LIN {X 0,Y 62.579,Z 548.254,A -85,B 0,C 180,E1 -28523.551,E2 -28523.551} C_VEL
LIN {X 0,Y 62.497,Z 549.862,A -85,B 0,C 180,E1 -28529.999,E2 -28529.999} C_VEL
LIN {X 0,Y 63.288,Z 551.85,A -85,B 0,C 180,E1 -28542.831,E2 -28542.831} C_VEL
LIN {X 0,Y 66.65,Z 552.168,A -85,B 0,C 180,E1 -28554.947,E2 -28554.947} C_VEL
LIN {X 0,Y 69.259,Z 551.826,A -85,B 0,C 180,E1 -28560.488,E2 -28560.488} C_VEL
LIN {X 0,Y 76.403,Z 549.954,A -85,B 0,C 180,E1 -28570.083,E2 -28570.083} C_VEL
LIN {X 0,Y 85.273,Z 546.396,A -85,B 0,C 180,E1 -28577.881,E2 -28577.881} C_VEL
LIN {X 0,Y 92.403,Z 542.869,A -85,B 0,C 180,E1 -28582.523,E2 -28582.523} C_VEL
LIN {X 0,Y 100.815,Z 537.874,A -85,B 0,C 180,E1 -28586.776,E2 -28586.776} C_VEL
LIN {X 0,Y 107.932,Z 532.997,A -85,B 0,C 180,E1 -28589.629,E2 -28589.629} C_VEL
LIN {X 0,Y 116.859,Z 525.752,A -85,B 0,C 180,E1 -28592.508,E2 -28592.508} C_VEL
LIN {X 0,Y 124.397,Z 518.518,A -85,B 0,C 180,E1 -28594.681,E2 -28594.681} C_VEL
LIN {X 0,Y 132.226,Z 509.719,A -85,B 0,C 180,E1 -28596.471,E2 -28596.471} C_VEL
LIN {X 0,Y 138.528,Z 501.33,A -85,B 0,C 180,E1 -28597.802,E2 -28597.802} C_VEL
LIN {X 0,Y 144.119,Z 492.584,A -85,B 0,C 180,E1 -28598.849,E2 -28598.849} C_VEL
LIN {X 0,Y 148.94,Z 483.625,A -85,B 0,C 180,E1 -28599.691,E2 -28599.691} C_VEL
LIN {X 0,Y 153.773,Z 472.412,A -85,B 0,C 180,E1 -28600.425,E2 -28600.425} C_VEL
LIN {X 0,Y 157.625,Z 460.628,A -85,B 0,C 180,E1 -28600.964,E2 -28600.964} C_VEL
LIN {X 0,Y 159.421,Z 453.709,A -85,B 0,C 180,E1 -28601.223,E2 -28601.223} C_VEL
LIN {X 0,Y 158.999,Z 451.366,A -85,B 0,C 180,E1 -28604.293,E2 -28604.293} C_VEL
LIN {X 0,Y 158.718,Z 450.737,A -85,B 0,C 180,E1 -28607.21,E2 -28607.21} C_VEL
LIN {X 0,Y 158.819,Z 450.724,A -85,B 0,C 180,E1 -28610.207,E2 -28610.207} C_VEL
LIN {X 0,Y 159.185,Z 451.615,A -85,B 0,C 180,E1 -28613.027,E2 -28613.027} C_VEL
LIN {X 0,Y 159.452,Z 453.17,A -85,B 0,C 180,E1 -28614.943,E2 -28614.943} C_VEL
LIN {X 0,Y 156.119,Z 465.329,A -85,B 0,C 180,E1 -28615.461,E2 -28615.461} C_VEL
LIN {X 0,Y 155.317,Z 467.61,A -85,B 0,C 180,E1 -28615.586,E2 -28615.586} C_VEL
LIN {X 0,Y 153.244,Z 473.27,A -85,B 0,C 180,E1 -28615.697,E2 -28615.697} C_VEL
LIN {X 0,Y 149.004,Z 482.069,A -85,B 0,C 180,E1 -28615.23,E2 -28615.23} C_VEL
LIN {X 0,Y 144.136,Z 490.614,A -85,B 0,C 180,E1 -28614.827,E2 -28614.827} C_VEL
LIN {X 0,Y 140.951,Z 495.515,A -85,B 0,C 180,E1 -28615.081,E2 -28615.081} C_VEL
LIN {X 0,Y 133.801,Z 505.556,A -85,B 0,C 180,E1 -28616.364,E2 -28616.364} C_VEL
LIN {X 0,Y 126.592,Z 514.036,A -85,B 0,C 180,E1 -28617.856,E2 -28617.856} C_VEL
LIN {X 0,Y 119.48,Z 521.172,A -85,B 0,C 180,E1 -28619.505,E2 -28619.505} C_VEL
LIN {X 0,Y 110.749,Z 528.549,A -85,B 0,C 180,E1 -28621.864,E2 -28621.864} C_VEL
LIN {X 0,Y 104.495,Z 533.192,A -85,B 0,C 180,E1 -28623.857,E2 -28623.857} C_VEL
LIN {X 0,Y 95.637,Z 538.703,A -85,B 0,C 180,E1 -28627.224,E2 -28627.224} C_VEL
LIN {X 0,Y 86.174,Z 543.493,A -85,B 0,C 180,E1 -28631.857,E2 -28631.857} C_VEL
LIN {X 0,Y 80.245,Z 546.021,A -85,B 0,C 180,E1 -28635.55,E2 -28635.55} C_VEL
LIN {X 0,Y 71.071,Z 549.044,A -85,B 0,C 180,E1 -28643.302,E2 -28643.302} C_VEL
LIN {X 0,Y 65.17,Z 550.355,A -85,B 0,C 180,E1 -28650.377,E2 -28650.377} C_VEL
LIN {X 0,Y 61.39,Z 550.71,A -85,B 0,C 180,E1 -28656.74,E2 -28656.74} C_VEL
LIN {X 0,Y 56.246,Z 550.229,A -85,B 0,C 180,E1 -28671.336,E2 -28671.336} C_VEL
LIN {X 0,Y 54.695,Z 548.382,A -85,B 0,C 180,E1 -28684.091,E2 -28684.091} C_VEL
LIN {X 0,Y 55.311,Z 545.786,A -85,B 0,C 180,E1 -28695.279,E2 -28695.279} C_VEL
LIN {X 0,Y 57.758,Z 541.882,A -85,B 0,C 180,E1 -28706.513,E2 -28706.513} C_VEL
LIN {X 0,Y 61.564,Z 536.786,A -85,B 0,C 180,E1 -28716.556,E2 -28716.556} C_VEL
LIN {X 0,Y 65.869,Z 531.542,A -85,B 0,C 180,E1 -28723.891,E2 -28723.891} C_VEL
LIN {X 0,Y 71.007,Z 525.185,A -85,B 0,C 180,E1 -28730.269,E2 -28730.269} C_VEL
LIN {X 0,Y 76.87,Z 517.465,A -85,B 0,C 180,E1 -28735.74,E2 -28735.74} C_VEL
LIN {X 0,Y 82.172,Z 509.761,A -85,B 0,C 180,E1 -28739.735,E2 -28739.735} C_VEL
LIN {X 0,Y 88.054,Z 500.156,A -85,B 0,C 180,E1 -28743.28,E2 -28743.28} C_VEL
LIN {X 0,Y 93,Z 490.72,A -85,B 0,C 180,E1 -28745.851,E2 -28745.851} C_VEL
LIN {X 0,Y 97.459,Z 480.559,A -85,B 0,C 180,E1 -28747.91,E2 -28747.91} C_VEL
LIN {X 0,Y 101.142,Z 470.239,A -85,B 0,C 180,E1 -28749.46,E2 -28749.46} C_VEL
LIN {X 0,Y 104.051,Z 459.662,A -85,B 0,C 180,E1 -28750.645,E2 -28750.645} C_VEL
LIN {X 0,Y 106.272,Z 449.078,A -85,B 0,C 180,E1 -28751.401,E2 -28751.401} C_VEL
LIN {X 0,Y 108.672,Z 430.245,A -85,B 0,C 180,E1 -28752.234,E2 -28752.234} C_VEL
LIN {X 0,Y 109.348,Z 423.381,A -85,B 0,C 180,E1 -28752.568,E2 -28752.568} C_VEL
LIN {X 0,Y 105.848,Z 414.809,A -85,B 0,C 180,E1 -28756.918,E2 -28756.918} C_VEL
LIN {X 0,Y 103.278,Z 409.54,A -85,B 0,C 180,E1 -28760.478,E2 -28760.478} C_VEL
LIN {X 0,Y 100.68,Z 404.348,A -85,B 0,C 180,E1 -28764.837,E2 -28764.837} C_VEL
LIN {X 0,Y 98.374,Z 400.234,A -85,B 0,C 180,E1 -28769.578,E2 -28769.578} C_VEL
LIN {X 0,Y 96.622,Z 396.989,A -85,B 0,C 180,E1 -28774.494,E2 -28774.494} C_VEL
LIN {X 0,Y 94.923,Z 393.92,A -85,B 0,C 180,E1 -28782.772,E2 -28782.772} C_VEL
LIN {X 0,Y 94.765,Z 392.903,A -85,B 0,C 180,E1 -28786.033,E2 -28786.033} C_VEL
LIN {X 0,Y 95.042,Z 392.871,A -85,B 0,C 180,E1 -28792.896,E2 -28792.896} C_VEL
LIN {X 0,Y 95.334,Z 393.924,A -85,B 0,C 180,E1 -28795.422,E2 -28795.422} C_VEL
LIN {X 0,Y 97.049,Z 397.206,A -85,B 0,C 180,E1 -28802.516,E2 -28802.516} C_VEL
LIN {X 0,Y 99.172,Z 401.426,A -85,B 0,C 180,E1 -28807.955,E2 -28807.955} C_VEL
LIN {X 0,Y 101.485,Z 405.932,A -85,B 0,C 180,E1 -28812.443,E2 -28812.443} C_VEL
LIN {X 0,Y 104.35,Z 411.648,A -85,B 0,C 180,E1 -28816.885,E2 -28816.885} C_VEL
LIN {X 0,Y 107.69,Z 419.475,A -85,B 0,C 180,E1 -28821.321,E2 -28821.321} C_VEL
LIN {X 0,Y 109.234,Z 424.676,A -85,B 0,C 180,E1 -28823.327,E2 -28823.327} C_VEL
LIN {X 0,Y 106.575,Z 448.2,A -85,B 0,C 180,E1 -28824.439,E2 -28824.439} C_VEL
LIN {X 0,Y 104.902,Z 457.507,A -85,B 0,C 180,E1 -28825.063,E2 -28825.063} C_VEL
LIN {X 0,Y 102.29,Z 467.768,A -85,B 0,C 180,E1 -28825.997,E2 -28825.997} C_VEL
LIN {X 0,Y 98.791,Z 478.018,A -85,B 0,C 180,E1 -28827.22,E2 -28827.22} C_VEL
LIN {X 0,Y 94.568,Z 488.531,A -85,B 0,C 180,E1 -28829.163,E2 -28829.163} C_VEL
LIN {X 0,Y 90.311,Z 497.107,A -85,B 0,C 180,E1 -28831.126,E2 -28831.126} C_VEL
LIN {X 0,Y 84.902,Z 506.569,A -85,B 0,C 180,E1 -28834.128,E2 -28834.128} C_VEL
LIN {X 0,Y 79.778,Z 514.509,A -85,B 0,C 180,E1 -28837.546,E2 -28837.546} C_VEL
LIN {X 0,Y 73.749,Z 522.723,A -85,B 0,C 180,E1 -28842.392,E2 -28842.392} C_VEL
LIN {X 0,Y 68.428,Z 529.57,A -85,B 0,C 180,E1 -28848.117,E2 -28848.117} C_VEL
LIN {X 0,Y 64.698,Z 534.284,A -85,B 0,C 180,E1 -28853.311,E2 -28853.311} C_VEL
LIN {X 0,Y 60.049,Z 540.007,A -85,B 0,C 180,E1 -28862.085,E2 -28862.085} C_VEL
LIN {X 0,Y 57.018,Z 544.501,A -85,B 0,C 180,E1 -28872.052,E2 -28872.052} C_VEL
LIN {X 0,Y 55.536,Z 547.885,A -85,B 0,C 180,E1 -28882.729,E2 -28882.729} C_VEL
LIN {X 0,Y 55.399,Z 549.494,A -85,B 0,C 180,E1 -28889.999,E2 -28889.999} C_VEL
LIN {X 0,Y 56.369,Z 551.641,A -85,B 0,C 180,E1 -28904.439,E2 -28904.439} C_VEL
LIN {X 0,Y 60.26,Z 552.123,A -85,B 0,C 180,E1 -28917.807,E2 -28917.807} C_VEL
LIN {X 0,Y 66.907,Z 551.075,A -85,B 0,C 180,E1 -28929.067,E2 -28929.067} C_VEL
LIN {X 0,Y 71.12,Z 550.096,A -85,B 0,C 180,E1 -28933.767,E2 -28933.767} C_VEL
LIN {X 0,Y 80.688,Z 546.707,A -85,B 0,C 180,E1 -28941.619,E2 -28941.619} C_VEL
LIN {X 0,Y 87.713,Z 543.606,A -85,B 0,C 180,E1 -28945.885,E2 -28945.885} C_VEL
LIN {X 0,Y 97.13,Z 538.467,A -85,B 0,C 180,E1 -28950.258,E2 -28950.258} C_VEL
LIN {X 0,Y 106.057,Z 532.618,A -85,B 0,C 180,E1 -28953.456,E2 -28953.456} C_VEL
LIN {X 0,Y 113.786,Z 526.723,A -85,B 0,C 180,E1 -28955.648,E2 -28955.648} C_VEL
LIN {X 0,Y 121.562,Z 519.697,A -85,B 0,C 180,E1 -28957.671,E2 -28957.671} C_VEL
LIN {X 0,Y 129.591,Z 511.148,A -85,B 0,C 180,E1 -28959.309,E2 -28959.309} C_VEL
LIN {X 0,Y 136.856,Z 501.867,A -85,B 0,C 180,E1 -28960.668,E2 -28960.668} C_VEL
LIN {X 0,Y 143.398,Z 491.794,A -85,B 0,C 180,E1 -28961.727,E2 -28961.727} C_VEL
LIN {X 0,Y 148.636,Z 482.026,A -85,B 0,C 180,E1 -28962.491,E2 -28962.491} C_VEL
LIN {X 0,Y 153.124,Z 471.638,A -85,B 0,C 180,E1 -28963.082,E2 -28963.082} C_VEL
LIN {X 0,Y 156.883,Z 460.246,A -85,B 0,C 180,E1 -28963.548,E2 -28963.548} C_VEL
LIN {X 0,Y 157.218,Z 458.926,A -85,B 0,C 180,E1 -28963.656,E2 -28963.656} C_VEL
LIN {X 0,Y 157.156,Z 458.077,A -85,B 0,C 180,E1 -28965.1,E2 -28965.1} C_VEL
LIN {X 0,Y 157.106,Z 457.5,A -85,B 0,C 180,E1 -28969.784,E2 -28969.784} C_VEL
LIN {X 0,Y 157.305,Z 458.378,A -85,B 0,C 180,E1 -28972.537,E2 -28972.537} C_VEL
LIN {X 0,Y 154.307,Z 468.079,A -85,B 0,C 180,E1 -28972.988,E2 -28972.988} C_VEL
LIN {X 0,Y 150.486,Z 477.718,A -85,B 0,C 180,E1 -28973.555,E2 -28973.555} C_VEL
LIN {X 0,Y 146.164,Z 486.6,A -85,B 0,C 180,E1 -28974.215,E2 -28974.215} C_VEL
LIN {X 0,Y 140.951,Z 495.515,A -85,B 0,C 180,E1 -28975.081,E2 -28975.081} C_VEL
LIN {X 0,Y 137.513,Z 500.486,A -85,B 0,C 180,E1 -28975.4,E2 -28975.4} C_VEL
LIN {X 0,Y 131.185,Z 508.137,A -85,B 0,C 180,E1 -28975.223,E2 -28975.223} C_VEL
LIN {X 0,Y 125.821,Z 513.891,A -85,B 0,C 180,E1 -28975.08,E2 -28975.08} C_VEL
LIN {X 0,Y 121.72,Z 517.927,A -85,B 0,C 180,E1 -28975.376,E2 -28975.376} C_VEL
LIN {X 0,Y 120.39,Z 519.235,A -85,B 0,C 180,E1 -28975.611,E2 -28975.611} C_VEL
LIN {X 0,Y 110.773,Z 527.458,A -85,B 0,C 180,E1 -28977.79,E2 -28977.79} C_VEL
LIN {X 0,Y 102.539,Z 533.342,A -85,B 0,C 180,E1 -28980.001,E2 -28980.001} C_VEL
LIN {X 0,Y 91.555,Z 539.688,A -85,B 0,C 180,E1 -28983.705,E2 -28983.705} C_VEL
LIN {X 0,Y 84.892,Z 542.977,A -85,B 0,C 180,E1 -28986.562,E2 -28986.562} C_VEL
LIN {X 0,Y 77.493,Z 545.911,A -85,B 0,C 180,E1 -28990.452,E2 -28990.452} C_VEL
LIN {X 0,Y 66.701,Z 549.19,A -85,B 0,C 180,E1 -28998.509,E2 -28998.509} C_VEL
LIN {X 0,Y 61.498,Z 550.225,A -85,B 0,C 180,E1 -29003.903,E2 -29003.903} C_VEL
LIN {X 0,Y 53.167,Z 550.86,A -85,B 0,C 180,E1 -29017.523,E2 -29017.523} C_VEL
LIN {X 0,Y 50.302,Z 550.478,A -85,B 0,C 180,E1 -29025.688,E2 -29025.688} C_VEL
LIN {X 0,Y 47.626,Z 548.209,A -85,B 0,C 180,E1 -29043.724,E2 -29043.724} C_VEL
LIN {X 0,Y 48.455,Z 545.257,A -85,B 0,C 180,E1 -29057.435,E2 -29057.435} C_VEL
LIN {X 0,Y 50.404,Z 542.497,A -85,B 0,C 180,E1 -29066.71,E2 -29066.71} C_VEL
LIN {X 0,Y 54.982,Z 536.889,A -85,B 0,C 180,E1 -29079.195,E2 -29079.195} C_VEL
LIN {X 0,Y 59.788,Z 531.572,A -85,B 0,C 180,E1 -29087.197,E2 -29087.197} C_VEL
LIN {X 0,Y 65.304,Z 525.296,A -85,B 0,C 180,E1 -29093.802,E2 -29093.802} C_VEL
LIN {X 0,Y 71.595,Z 517.585,A -85,B 0,C 180,E1 -29099.395,E2 -29099.395} C_VEL
LIN {X 0,Y 77.65,Z 509.248,A -85,B 0,C 180,E1 -29103.668,E2 -29103.668} C_VEL
LIN {X 0,Y 83.432,Z 500.296,A -85,B 0,C 180,E1 -29106.884,E2 -29106.884} C_VEL
LIN {X 0,Y 88.629,Z 490.865,A -85,B 0,C 180,E1 -29109.374,E2 -29109.374} C_VEL
LIN {X 0,Y 93.319,Z 480.637,A -85,B 0,C 180,E1 -29111.367,E2 -29111.367} C_VEL
LIN {X 0,Y 97.129,Z 470.418,A -85,B 0,C 180,E1 -29112.831,E2 -29112.831} C_VEL
LIN {X 0,Y 100.176,Z 459.798,A -85,B 0,C 180,E1 -29113.966,E2 -29113.966} C_VEL
LIN {X 0,Y 102.53,Z 448.814,A -85,B 0,C 180,E1 -29114.707,E2 -29114.707} C_VEL
LIN {X 0,Y 105.009,Z 429.995,A -85,B 0,C 180,E1 -29115.479,E2 -29115.479} C_VEL
LIN {X 0,Y 105.349,Z 426.176,A -85,B 0,C 180,E1 -29115.714,E2 -29115.714} C_VEL
LIN {X 0,Y 102.535,Z 419.019,A -85,B 0,C 180,E1 -29119.721,E2 -29119.721} C_VEL
LIN {X 0,Y 100.478,Z 414.401,A -85,B 0,C 180,E1 -29123.086,E2 -29123.086} C_VEL
LIN {X 0,Y 98.288,Z 409.831,A -85,B 0,C 180,E1 -29127.354,E2 -29127.354} C_VEL
LIN {X 0,Y 96.71,Z 406.687,A -85,B 0,C 180,E1 -29131.104,E2 -29131.104} C_VEL
LIN {X 0,Y 95.41,Z 403.865,A -85,B 0,C 180,E1 -29135.269,E2 -29135.269} C_VEL
LIN {X 0,Y 93.898,Z 400.897,A -85,B 0,C 180,E1 -29143.485,E2 -29143.485} C_VEL
LIN {X 0,Y 93.812,Z 399.843,A -85,B 0,C 180,E1 -29146.885,E2 -29146.885} C_VEL
LIN {X 0,Y 94.088,Z 399.927,A -85,B 0,C 180,E1 -29152.824,E2 -29152.824} C_VEL
LIN {X 0,Y 95.437,Z 403.356,A -85,B 0,C 180,E1 -29160.438,E2 -29160.438} C_VEL
LIN {X 0,Y 97.386,Z 407.758,A -85,B 0,C 180,E1 -29166.36,E2 -29166.36} C_VEL
LIN {X 0,Y 99.483,Z 412.149,A -85,B 0,C 180,E1 -29170.87,E2 -29170.87} C_VEL
LIN {X 0,Y 101.983,Z 417.768,A -85,B 0,C 180,E1 -29175.248,E2 -29175.248} C_VEL
LIN {X 0,Y 104.852,Z 425.115,A -85,B 0,C 180,E1 -29179.474,E2 -29179.474} C_VEL
LIN {X 0,Y 105.33,Z 427.034,A -85,B 0,C 180,E1 -29180.221,E2 -29180.221} C_VEL
LIN {X 0,Y 102.71,Z 448.613,A -85,B 0,C 180,E1 -29181.177,E2 -29181.177} C_VEL
LIN {X 0,Y 100.863,Z 458.234,A -85,B 0,C 180,E1 -29181.812,E2 -29181.812} C_VEL
LIN {X 0,Y 98.478,Z 467.269,A -85,B 0,C 180,E1 -29182.585,E2 -29182.585} C_VEL
LIN {X 0,Y 94.984,Z 477.329,A -85,B 0,C 180,E1 -29183.701,E2 -29183.701} C_VEL
LIN {X 0,Y 90.554,Z 487.949,A -85,B 0,C 180,E1 -29185.546,E2 -29185.546} C_VEL
LIN {X 0,Y 85.351,Z 497.835,A -85,B 0,C 180,E1 -29187.725,E2 -29187.725} C_VEL
LIN {X 0,Y 80.408,Z 506.141,A -85,B 0,C 180,E1 -29190.331,E2 -29190.331} C_VEL
LIN {X 0,Y 74.669,Z 514.521,A -85,B 0,C 180,E1 -29193.895,E2 -29193.895} C_VEL
LIN {X 0,Y 69.115,Z 521.673,A -85,B 0,C 180,E1 -29197.994,E2 -29197.994} C_VEL
LIN {X 0,Y 63.283,Z 528.687,A -85,B 0,C 180,E1 -29203.79,E2 -29203.79} C_VEL
LIN {X 0,Y 57.179,Z 535.494,A -85,B 0,C 180,E1 -29212.079,E2 -29212.079} C_VEL
LIN {X 0,Y 53.834,Z 539.341,A -85,B 0,C 180,E1 -29218.519,E2 -29218.519} C_VEL
LIN {X 0,Y 50.305,Z 543.975,A -85,B 0,C 180,E1 -29229.556,E2 -29229.556} C_VEL
LIN {X 0,Y 48.498,Z 547.462,A -85,B 0,C 180,E1 -29241.667,E2 -29241.667} C_VEL
LIN {X 0,Y 48.316,Z 549.117,A -85,B 0,C 180,E1 -29249.999,E2 -29249.999} C_VEL
LIN {X 0,Y 48.527,Z 550.457,A -85,B 0,C 180,E1 -29258.326,E2 -29258.326} C_VEL
LIN {X 0,Y 49.517,Z 551.373,A -85,B 0,C 180,E1 -29266.49,E2 -29266.49} C_VEL
LIN {X 0,Y 54.062,Z 552.07,A -85,B 0,C 180,E1 -29281.331,E2 -29281.331} C_VEL
LIN {X 0,Y 61.542,Z 551.147,A -85,B 0,C 180,E1 -29293.25,E2 -29293.25} C_VEL
LIN {X 0,Y 66.178,Z 550.179,A -85,B 0,C 180,E1 -29298.02,E2 -29298.02} C_VEL
LIN {X 0,Y 76.489,Z 547.032,A -85,B 0,C 180,E1 -29305.785,E2 -29305.785} C_VEL
LIN {X 0,Y 84.622,Z 543.711,A -85,B 0,C 180,E1 -29310.213,E2 -29310.213} C_VEL
LIN {X 0,Y 93.834,Z 539.073,A -85,B 0,C 180,E1 -29313.998,E2 -29313.998} C_VEL
LIN {X 0,Y 104.694,Z 532.251,A -85,B 0,C 180,E1 -29317.371,E2 -29317.371} C_VEL
LIN {X 0,Y 112.665,Z 526.309,A -85,B 0,C 180,E1 -29319.34,E2 -29319.34} C_VEL
LIN {X 0,Y 120.7,Z 519.228,A -85,B 0,C 180,E1 -29321.118,E2 -29321.118} C_VEL
LIN {X 0,Y 128.936,Z 510.63,A -85,B 0,C 180,E1 -29322.531,E2 -29322.531} C_VEL
LIN {X 0,Y 136.368,Z 501.3,A -85,B 0,C 180,E1 -29323.713,E2 -29323.713} C_VEL
LIN {X 0,Y 142.207,Z 492.611,A -85,B 0,C 180,E1 -29324.517,E2 -29324.517} C_VEL
LIN {X 0,Y 147.413,Z 483.333,A -85,B 0,C 180,E1 -29325.169,E2 -29325.169} C_VEL
LIN {X 0,Y 152.298,Z 472.444,A -85,B 0,C 180,E1 -29325.713,E2 -29325.713} C_VEL
LIN {X 0,Y 154.656,Z 465.985,A -85,B 0,C 180,E1 -29325.948,E2 -29325.948} C_VEL
LIN {X 0,Y 155.112,Z 464.655,A -85,B 0,C 180,E1 -29326.24,E2 -29326.24} C_VEL
LIN {X 0,Y 155.153,Z 464.327,A -85,B 0,C 180,E1 -29329.562,E2 -29329.562} C_VEL
LIN {X 0,Y 155.046,Z 464.786,A -85,B 0,C 180,E1 -29330.214,E2 -29330.214} C_VEL
LIN {X 0,Y 150.759,Z 476.023,A -85,B 0,C 180,E1 -29330.751,E2 -29330.751} C_VEL
LIN {X 0,Y 145.577,Z 486.601,A -85,B 0,C 180,E1 -29331.414,E2 -29331.414} C_VEL
LIN {X 0,Y 139.17,Z 497.084,A -85,B 0,C 180,E1 -29332.327,E2 -29332.327} C_VEL
LIN {X 0,Y 133.168,Z 505.297,A -85,B 0,C 180,E1 -29333.251,E2 -29333.251} C_VEL
LIN {X 0,Y 127.13,Z 512.444,A -85,B 0,C 180,E1 -29334.308,E2 -29334.308} C_VEL
LIN {X 0,Y 120.39,Z 519.235,A -85,B 0,C 180,E1 -29335.611,E2 -29335.611} C_VEL
LIN {X 0,Y 116.103,Z 523.127,A -85,B 0,C 180,E1 -29336.187,E2 -29336.187} C_VEL
LIN {X 0,Y 108.162,Z 529.063,A -85,B 0,C 180,E1 -29336.398,E2 -29336.398} C_VEL
LIN {X 0,Y 99.786,Z 534.345,A -85,B 0,C 180,E1 -29336.751,E2 -29336.751} C_VEL
LIN {X 0,Y 94.843,Z 537.103,A -85,B 0,C 180,E1 -29337.684,E2 -29337.684} C_VEL
LIN {X 0,Y 84.353,Z 542.331,A -85,B 0,C 180,E1 -29341.161,E2 -29341.161} C_VEL
LIN {X 0,Y 74.678,Z 546.087,A -85,B 0,C 180,E1 -29345.401,E2 -29345.401} C_VEL
LIN {X 0,Y 63.066,Z 549.311,A -85,B 0,C 180,E1 -29352.88,E2 -29352.88} C_VEL
LIN {X 0,Y 52.785,Z 550.796,A -85,B 0,C 180,E1 -29363.545,E2 -29363.545} C_VEL
LIN {X 0,Y 48.701,Z 551.043,A -85,B 0,C 180,E1 -29370.021,E2 -29370.021} C_VEL
LIN {X 0,Y 44.851,Z 550.667,A -85,B 0,C 180,E1 -29378.816,E2 -29378.816} C_VEL
LIN {X 0,Y 40.748,Z 548.75,A -85,B 0,C 180,E1 -29398.842,E2 -29398.842} C_VEL
LIN {X 0,Y 40.946,Z 545.976,A -85,B 0,C 180,E1 -29415.081,E2 -29415.081} C_VEL
LIN {X 0,Y 43.823,Z 542.062,A -85,B 0,C 180,E1 -29430.001,E2 -29430.001} C_VEL
LIN {X 0,Y 48.566,Z 536.955,A -85,B 0,C 180,E1 -29442.538,E2 -29442.538} C_VEL
LIN {X 0,Y 54.925,Z 530.478,A -85,B 0,C 180,E1 -29452.574,E2 -29452.574} C_VEL
LIN {X 0,Y 59.878,Z 525.348,A -85,B 0,C 180,E1 -29458.002,E2 -29458.002} C_VEL
LIN {X 0,Y 66.248,Z 518.135,A -85,B 0,C 180,E1 -29463.322,E2 -29463.322} C_VEL
LIN {X 0,Y 73.09,Z 509.278,A -85,B 0,C 180,E1 -29467.807,E2 -29467.807} C_VEL
LIN {X 0,Y 79.188,Z 500.313,A -85,B 0,C 180,E1 -29470.885,E2 -29470.885} C_VEL
LIN {X 0,Y 84.634,Z 490.868,A -85,B 0,C 180,E1 -29473.243,E2 -29473.243} C_VEL
LIN {X 0,Y 89.35,Z 481.023,A -85,B 0,C 180,E1 -29475.066,E2 -29475.066} C_VEL
LIN {X 0,Y 93.445,Z 470.488,A -85,B 0,C 180,E1 -29476.473,E2 -29476.473} C_VEL
LIN {X 0,Y 96.551,Z 460.069,A -85,B 0,C 180,E1 -29477.527,E2 -29477.527} C_VEL
LIN {X 0,Y 98.918,Z 449.563,A -85,B 0,C 180,E1 -29478.196,E2 -29478.196} C_VEL
LIN {X 0,Y 101.414,Z 431.476,A -85,B 0,C 180,E1 -29478.897,E2 -29478.897} C_VEL
LIN {X 0,Y 101.641,Z 429.062,A -85,B 0,C 180,E1 -29479.046,E2 -29479.046} C_VEL
LIN {X 0,Y 99.037,Z 421.97,A -85,B 0,C 180,E1 -29483.562,E2 -29483.562} C_VEL
LIN {X 0,Y 96.676,Z 416.478,A -85,B 0,C 180,E1 -29488.517,E2 -29488.517} C_VEL
LIN {X 0,Y 95.249,Z 413.337,A -85,B 0,C 180,E1 -29492.305,E2 -29492.305} C_VEL
LIN {X 0,Y 94.029,Z 410.53,A -85,B 0,C 180,E1 -29496.773,E2 -29496.773} C_VEL
LIN {X 0,Y 92.868,Z 406.913,A -85,B 0,C 180,E1 -29506.876,E2 -29506.876} C_VEL
LIN {X 0,Y 93.062,Z 406.886,A -85,B 0,C 180,E1 -29512.029,E2 -29512.029} C_VEL
LIN {X 0,Y 94.309,Z 410.583,A -85,B 0,C 180,E1 -29519.999,E2 -29519.999} C_VEL
LIN {X 0,Y 95.781,Z 414.352,A -85,B 0,C 180,E1 -29524.997,E2 -29524.997} C_VEL
LIN {X 0,Y 97.889,Z 419.157,A -85,B 0,C 180,E1 -29529.955,E2 -29529.955} C_VEL
LIN {X 0,Y 99.814,Z 424.238,A -85,B 0,C 180,E1 -29533.746,E2 -29533.746} C_VEL
LIN {X 0,Y 101.681,Z 429.474,A -85,B 0,C 180,E1 -29536.886,E2 -29536.886} C_VEL
LIN {X 0,Y 99.239,Z 448.532,A -85,B 0,C 180,E1 -29537.674,E2 -29537.674} C_VEL
LIN {X 0,Y 97.459,Z 457.592,A -85,B 0,C 180,E1 -29538.222,E2 -29538.222} C_VEL
LIN {X 0,Y 94.774,Z 467.443,A -85,B 0,C 180,E1 -29539.004,E2 -29539.004} C_VEL
LIN {X 0,Y 91.563,Z 476.503,A -85,B 0,C 180,E1 -29539.904,E2 -29539.904} C_VEL
LIN {X 0,Y 86.933,Z 487.254,A -85,B 0,C 180,E1 -29541.61,E2 -29541.61} C_VEL
LIN {X 0,Y 81.513,Z 497.241,A -85,B 0,C 180,E1 -29543.639,E2 -29543.639} C_VEL
LIN {X 0,Y 75.583,Z 506.661,A -85,B 0,C 180,E1 -29546.494,E2 -29546.494} C_VEL
LIN {X 0,Y 70.526,Z 513.682,A -85,B 0,C 180,E1 -29549.316,E2 -29549.316} C_VEL
LIN {X 0,Y 63.391,Z 522.283,A -85,B 0,C 180,E1 -29554.303,E2 -29554.303} C_VEL
LIN {X 0,Y 57.354,Z 528.933,A -85,B 0,C 180,E1 -29560.016,E2 -29560.016} C_VEL
LIN {X 0,Y 51.755,Z 534.711,A -85,B 0,C 180,E1 -29567.235,E2 -29567.235} C_VEL
LIN {X 0,Y 46.294,Z 540.287,A -85,B 0,C 180,E1 -29577.903,E2 -29577.903} C_VEL
LIN {X 0,Y 42.738,Z 544.658,A -85,B 0,C 180,E1 -29590.798,E2 -29590.798} C_VEL
LIN {X 0,Y 41.497,Z 546.964,A -85,B 0,C 180,E1 -29600.248,E2 -29600.248} C_VEL
LIN {X 0,Y 41.227,Z 548.729,A -85,B 0,C 180,E1 -29609.999,E2 -29609.999} C_VEL
LIN {X 0,Y 41.516,Z 550.185,A -85,B 0,C 180,E1 -29619.745,E2 -29619.745} C_VEL
LIN {X 0,Y 45.011,Z 551.678,A -85,B 0,C 180,E1 -29637.931,E2 -29637.931} C_VEL
LIN {X 0,Y 48.108,Z 551.958,A -85,B 0,C 180,E1 -29645.757,E2 -29645.757} C_VEL
LIN {X 0,Y 56.57,Z 551.228,A -85,B 0,C 180,E1 -29658.194,E2 -29658.194} C_VEL
LIN {X 0,Y 67.037,Z 548.939,A -85,B 0,C 180,E1 -29667.003,E2 -29667.003} C_VEL
LIN {X 0,Y 75.676,Z 546.236,A -85,B 0,C 180,E1 -29671.916,E2 -29671.916} C_VEL
LIN {X 0,Y 84.685,Z 542.58,A -85,B 0,C 180,E1 -29675.907,E2 -29675.907} C_VEL
LIN {X 0,Y 94.146,Z 537.845,A -85,B 0,C 180,E1 -29678.927,E2 -29678.927} C_VEL
LIN {X 0,Y 103.823,Z 531.919,A -85,B 0,C 180,E1 -29681.385,E2 -29681.385} C_VEL
LIN {X 0,Y 112.005,Z 525.966,A -85,B 0,C 180,E1 -29683.114,E2 -29683.114} C_VEL
LIN {X 0,Y 120.291,Z 518.833,A -85,B 0,C 180,E1 -29684.582,E2 -29684.582} C_VEL
LIN {X 0,Y 128.693,Z 510.179,A -85,B 0,C 180,E1 -29685.775,E2 -29685.775} C_VEL
LIN {X 0,Y 135.43,Z 501.96,A -85,B 0,C 180,E1 -29686.657,E2 -29686.657} C_VEL
LIN {X 0,Y 142.211,Z 491.979,A -85,B 0,C 180,E1 -29687.431,E2 -29687.431} C_VEL
LIN {X 0,Y 146.303,Z 484.969,A -85,B 0,C 180,E1 -29687.874,E2 -29687.874} C_VEL
LIN {X 0,Y 147.001,Z 483.596,A -85,B 0,C 180,E1 -29688.437,E2 -29688.437} C_VEL
LIN {X 0,Y 139.474,Z 496.193,A -85,B 0,C 180,E1 -29689.292,E2 -29689.292} C_VEL
LIN {X 0,Y 132.996,Z 505.003,A -85,B 0,C 180,E1 -29690.124,E2 -29690.124} C_VEL
LIN {X 0,Y 126.265,Z 512.778,A -85,B 0,C 180,E1 -29691.105,E2 -29691.105} C_VEL
LIN {X 0,Y 117.471,Z 521.215,A -85,B 0,C 180,E1 -29692.552,E2 -29692.552} C_VEL
LIN {X 0,Y 109.513,Z 527.695,A -85,B 0,C 180,E1 -29694.101,E2 -29694.101} C_VEL
LIN {X 0,Y 101.046,Z 533.526,A -85,B 0,C 180,E1 -29696.013,E2 -29696.013} C_VEL
LIN {X 0,Y 94.843,Z 537.103,A -85,B 0,C 180,E1 -29697.684,E2 -29697.684} C_VEL
LIN {X 0,Y 89.804,Z 539.736,A -85,B 0,C 180,E1 -29698.766,E2 -29698.766} C_VEL
LIN {X 0,Y 77.043,Z 544.868,A -85,B 0,C 180,E1 -29700.105,E2 -29700.105} C_VEL
LIN {X 0,Y 69.714,Z 547.112,A -85,B 0,C 180,E1 -29701.558,E2 -29701.558} C_VEL
LIN {X 0,Y 66.288,Z 547.969,A -85,B 0,C 180,E1 -29702.97,E2 -29702.97} C_VEL
LIN {X 0,Y 56.914,Z 549.943,A -85,B 0,C 180,E1 -29708.936,E2 -29708.936} C_VEL
LIN {X 0,Y 48.576,Z 550.912,A -85,B 0,C 180,E1 -29716.822,E2 -29716.822} C_VEL
LIN {X 0,Y 45.232,Z 551.111,A -85,B 0,C 180,E1 -29721.212,E2 -29721.212} C_VEL
LIN {X 0,Y 39.24,Z 550.761,A -85,B 0,C 180,E1 -29732.503,E2 -29732.503} C_VEL
LIN {X 0,Y 34.257,Z 549.185,A -85,B 0,C 180,E1 -29752.016,E2 -29752.016} C_VEL
LIN {X 0,Y 33.54,Z 546.611,A -85,B 0,C 180,E1 -29771.682,E2 -29771.682} C_VEL
LIN {X 0,Y 36.235,Z 542.918,A -85,B 0,C 180,E1 -29790.001,E2 -29790.001} C_VEL
LIN {X 0,Y 42.365,Z 537.022,A -85,B 0,C 180,E1 -29806.877,E2 -29806.877} C_VEL
LIN {X 0,Y 48.191,Z 531.765,A -85,B 0,C 180,E1 -29815.946,E2 -29815.946} C_VEL
LIN {X 0,Y 54.859,Z 525.394,A -85,B 0,C 180,E1 -29822.989,E2 -29822.989} C_VEL
LIN {X 0,Y 61.807,Z 518.049,A -85,B 0,C 180,E1 -29828.258,E2 -29828.258} C_VEL
LIN {X 0,Y 68.961,Z 509.307,A -85,B 0,C 180,E1 -29832.468,E2 -29832.468} C_VEL
LIN {X 0,Y 75.38,Z 500.32,A -85,B 0,C 180,E1 -29835.31,E2 -29835.31} C_VEL
LIN {X 0,Y 81.063,Z 490.856,A -85,B 0,C 180,E1 -29837.472,E2 -29837.472} C_VEL
LIN {X 0,Y 85.942,Z 481.019,A -85,B 0,C 180,E1 -29839.139,E2 -29839.139} C_VEL
LIN {X 0,Y 89.635,Z 472.089,A -85,B 0,C 180,E1 -29840.25,E2 -29840.25} C_VEL
LIN {X 0,Y 93.458,Z 459.787,A -85,B 0,C 180,E1 -29841.373,E2 -29841.373} C_VEL
LIN {X 0,Y 95.85,Z 449.4,A -85,B 0,C 180,E1 -29841.944,E2 -29841.944} C_VEL
LIN {X 0,Y 98.282,Z 432.214,A -85,B 0,C 180,E1 -29842.565,E2 -29842.565} C_VEL
LIN {X 0,Y 96.566,Z 427.159,A -85,B 0,C 180,E1 -29846.162,E2 -29846.162} C_VEL
LIN {X 0,Y 94.848,Z 422.622,A -85,B 0,C 180,E1 -29850.374,E2 -29850.374} C_VEL
LIN {X 0,Y 93.622,Z 419.544,A -85,B 0,C 180,E1 -29854.267,E2 -29854.267} C_VEL
LIN {X 0,Y 92.661,Z 417.127,A -85,B 0,C 180,E1 -29858.434,E2 -29858.434} C_VEL
LIN {X 0,Y 91.916,Z 414.062,A -85,B 0,C 180,E1 -29866.738,E2 -29866.738} C_VEL
LIN {X 0,Y 92.071,Z 414.025,A -85,B 0,C 180,E1 -29871.675,E2 -29871.675} C_VEL
LIN {X 0,Y 93.004,Z 417.257,A -85,B 0,C 180,E1 -29878.671,E2 -29878.671} C_VEL
LIN {X 0,Y 94.255,Z 420.935,A -85,B 0,C 180,E1 -29883.643,E2 -29883.643} C_VEL
LIN {X 0,Y 96.158,Z 425.968,A -85,B 0,C 180,E1 -29888.719,E2 -29888.719} C_VEL
LIN {X 0,Y 97.855,Z 431.033,A -85,B 0,C 180,E1 -29892.442,E2 -29892.442} C_VEL
LIN {X 0,Y 98.291,Z 432.464,A -85,B 0,C 180,E1 -29893.322,E2 -29893.322} C_VEL
LIN {X 0,Y 95.858,Z 450.133,A -85,B 0,C 180,E1 -29894.01,E2 -29894.01} C_VEL
LIN {X 0,Y 92.915,Z 462.886,A -85,B 0,C 180,E1 -29894.739,E2 -29894.739} C_VEL
LIN {X 0,Y 88.547,Z 475.685,A -85,B 0,C 180,E1 -29895.837,E2 -29895.837} C_VEL
LIN {X 0,Y 83.756,Z 486.518,A -85,B 0,C 180,E1 -29897.352,E2 -29897.352} C_VEL
LIN {X 0,Y 78.129,Z 496.622,A -85,B 0,C 180,E1 -29899.174,E2 -29899.174} C_VEL
LIN {X 0,Y 71.903,Z 506.129,A -85,B 0,C 180,E1 -29901.788,E2 -29901.788} C_VEL
LIN {X 0,Y 65.82,Z 514.086,A -85,B 0,C 180,E1 -29904.831,E2 -29904.831} C_VEL
LIN {X 0,Y 59.32,Z 521.473,A -85,B 0,C 180,E1 -29908.806,E2 -29908.806} C_VEL
LIN {X 0,Y 51.735,Z 529.178,A -85,B 0,C 180,E1 -29915.403,E2 -29915.403} C_VEL
LIN {X 0,Y 46.786,Z 533.896,A -85,B 0,C 180,E1 -29921.315,E2 -29921.315} C_VEL
LIN {X 0,Y 40.43,Z 539.639,A -85,B 0,C 180,E1 -29932.524,E2 -29932.524} C_VEL
LIN {X 0,Y 36.085,Z 544.144,A -85,B 0,C 180,E1 -29947.074,E2 -29947.074} C_VEL
LIN {X 0,Y 34.519,Z 546.453,A -85,B 0,C 180,E1 -29958.251,E2 -29958.251} C_VEL
LIN {X 0,Y 34.126,Z 548.34,A -85,B 0,C 180,E1 -29969.999,E2 -29969.999} C_VEL
LIN {X 0,Y 34.533,Z 549.881,A -85,B 0,C 180,E1 -29981.741,E2 -29981.741} C_VEL
LIN {X 0,Y 38.851,Z 551.517,A -85,B 0,C 180,E1 -30002.865,E2 -30002.865} C_VEL
LIN {X 0,Y 42.521,Z 551.798,A -85,B 0,C 180,E1 -30011.385,E2 -30011.385} C_VEL
LIN {X 0,Y 52.1,Z 551.29,A -85,B 0,C 180,E1 -30024.032,E2 -30024.032} C_VEL
LIN {X 0,Y 63.447,Z 549.149,A -85,B 0,C 180,E1 -30032.394,E2 -30032.394} C_VEL
LIN {X 0,Y 73.709,Z 546.18,A -85,B 0,C 180,E1 -30037.36,E2 -30037.36} C_VEL
LIN {X 0,Y 82.051,Z 543.087,A -85,B 0,C 180,E1 -30040.421,E2 -30040.421} C_VEL
LIN {X 0,Y 91.848,Z 538.52,A -85,B 0,C 180,E1 -30043.032,E2 -30043.032} C_VEL
LIN {X 0,Y 101.796,Z 532.769,A -85,B 0,C 180,E1 -30045.14,E2 -30045.14} C_VEL
LIN {X 0,Y 111.855,Z 525.627,A -85,B 0,C 180,E1 -30046.877,E2 -30046.877} C_VEL
LIN {X 0,Y 120.325,Z 518.436,A -85,B 0,C 180,E1 -30048.052,E2 -30048.052} C_VEL
LIN {X 0,Y 122.033,Z 516.769,A -85,B 0,C 180,E1 -30048.25,E2 -30048.25} C_VEL
LIN {X 0,Y 116.095,Z 522.115,A -85,B 0,C 180,E1 -30049.169,E2 -30049.169} C_VEL
LIN {X 0,Y 108.715,Z 527.95,A -85,B 0,C 180,E1 -30050.351,E2 -30050.351} C_VEL
LIN {X 0,Y 97.475,Z 535.18,A -85,B 0,C 180,E1 -30052.47,E2 -30052.47} C_VEL
LIN {X 0,Y 88.626,Z 539.858,A -85,B 0,C 180,E1 -30054.61,E2 -30054.61} C_VEL
LIN {X 0,Y 80.941,Z 543.293,A -85,B 0,C 180,E1 -30056.887,E2 -30056.887} C_VEL
LIN {X 0,Y 70.29,Z 546.951,A -85,B 0,C 180,E1 -30060.986,E2 -30060.986} C_VEL
LIN {X 0,Y 66.288,Z 547.969,A -85,B 0,C 180,E1 -30062.97,E2 -30062.97} C_VEL
LIN {X 0,Y 61.078,Z 549.241,A -85,B 0,C 180,E1 -30065.26,E2 -30065.26} C_VEL
LIN {X 0,Y 51.732,Z 550.613,A -85,B 0,C 180,E1 -30068.36,E2 -30068.36} C_VEL
LIN {X 0,Y 44.287,Z 551.079,A -85,B 0,C 180,E1 -30071.652,E2 -30071.652} C_VEL
LIN {X 0,Y 39.246,Z 551.206,A -85,B 0,C 180,E1 -30075.916,E2 -30075.916} C_VEL
LIN {X 0,Y 37.791,Z 551.075,A -85,B 0,C 180,E1 -30077.898,E2 -30077.898} C_VEL
LIN {X 0,Y 32.188,Z 550.617,A -85,B 0,C 180,E1 -30089.148,E2 -30089.148} C_VEL
LIN {X 0,Y 27.095,Z 548.774,A -85,B 0,C 180,E1 -30111.096,E2 -30111.096} C_VEL
LIN {X 0,Y 26.588,Z 546.116,A -85,B 0,C 180,E1 -30134.675,E2 -30134.675} C_VEL
LIN {X 0,Y 30.198,Z 542.181,A -85,B 0,C 180,E1 -30156.684,E2 -30156.684} C_VEL
LIN {X 0,Y 36.485,Z 537.047,A -85,B 0,C 180,E1 -30172.661,E2 -30172.661} C_VEL
LIN {X 0,Y 43.014,Z 531.782,A -85,B 0,C 180,E1 -30182.075,E2 -30182.075} C_VEL
LIN {X 0,Y 50.323,Z 525.397,A -85,B 0,C 180,E1 -30188.938,E2 -30188.938} C_VEL
LIN {X 0,Y 58.291,Z 517.47,A -85,B 0,C 180,E1 -30194.132,E2 -30194.132} C_VEL
LIN {X 0,Y 65.352,Z 509.281,A -85,B 0,C 180,E1 -30197.676,E2 -30197.676} C_VEL
LIN {X 0,Y 72.059,Z 500.279,A -85,B 0,C 180,E1 -30200.181,E2 -30200.181} C_VEL
LIN {X 0,Y 77.959,Z 490.797,A -85,B 0,C 180,E1 -30202.076,E2 -30202.076} C_VEL
LIN {X 0,Y 82.486,Z 482.125,A -85,B 0,C 180,E1 -30203.385,E2 -30203.385} C_VEL
LIN {X 0,Y 87.066,Z 471.266,A -85,B 0,C 180,E1 -30204.539,E2 -30204.539} C_VEL
LIN {X 0,Y 90.686,Z 459.921,A -85,B 0,C 180,E1 -30205.429,E2 -30205.429} C_VEL
LIN {X 0,Y 93.102,Z 449.729,A -85,B 0,C 180,E1 -30205.922,E2 -30205.922} C_VEL
LIN {X 0,Y 95.229,Z 435.314,A -85,B 0,C 180,E1 -30206.443,E2 -30206.443} C_VEL
LIN {X 0,Y 93.572,Z 430.017,A -85,B 0,C 180,E1 -30210.897,E2 -30210.897} C_VEL
LIN {X 0,Y 92.161,Z 425.914,A -85,B 0,C 180,E1 -30216.045,E2 -30216.045} C_VEL
LIN {X 0,Y 91.448,Z 423.887,A -85,B 0,C 180,E1 -30219.688,E2 -30219.688} C_VEL
LIN {X 0,Y 90.975,Z 421.026,A -85,B 0,C 180,E1 -30227.864,E2 -30227.864} C_VEL
LIN {X 0,Y 91.079,Z 421.316,A -85,B 0,C 180,E1 -30231.495,E2 -30231.495} C_VEL
LIN {X 0,Y 91.745,Z 423.985,A -85,B 0,C 180,E1 -30237.417,E2 -30237.417} C_VEL
LIN {X 0,Y 92.774,Z 427.533,A -85,B 0,C 180,E1 -30242.225,E2 -30242.225} C_VEL
LIN {X 0,Y 94.379,Z 432.498,A -85,B 0,C 180,E1 -30247.216,E2 -30247.216} C_VEL
LIN {X 0,Y 95.262,Z 435.639,A -85,B 0,C 180,E1 -30249.501,E2 -30249.501} C_VEL
LIN {X 0,Y 92.952,Z 451.377,A -85,B 0,C 180,E1 -30250.088,E2 -30250.088} C_VEL
LIN {X 0,Y 89.245,Z 465.815,A -85,B 0,C 180,E1 -30250.904,E2 -30250.904} C_VEL
LIN {X 0,Y 85.221,Z 476.57,A -85,B 0,C 180,E1 -30251.672,E2 -30251.672} C_VEL
LIN {X 0,Y 80.251,Z 487.266,A -85,B 0,C 180,E1 -30253.022,E2 -30253.022} C_VEL
LIN {X 0,Y 74.426,Z 497.193,A -85,B 0,C 180,E1 -30254.554,E2 -30254.554} C_VEL
LIN {X 0,Y 68.759,Z 505.566,A -85,B 0,C 180,E1 -30256.616,E2 -30256.616} C_VEL
LIN {X 0,Y 61.585,Z 514.456,A -85,B 0,C 180,E1 -30259.697,E2 -30259.697} C_VEL
LIN {X 0,Y 53.848,Z 522.608,A -85,B 0,C 180,E1 -30263.989,E2 -30263.989} C_VEL
LIN {X 0,Y 46.542,Z 529.396,A -85,B 0,C 180,E1 -30269.74,E2 -30269.74} C_VEL
LIN {X 0,Y 39.8,Z 535.044,A -85,B 0,C 180,E1 -30277.378,E2 -30277.378} C_VEL
LIN {X 0,Y 32.98,Z 540.504,A -85,B 0,C 180,E1 -30290.259,E2 -30290.259} C_VEL
LIN {X 0,Y 28.462,Z 544.765,A -85,B 0,C 180,E1 -30308.258,E2 -30308.258} C_VEL
LIN {X 0,Y 27.031,Z 547.931,A -85,B 0,C 180,E1 -30329.998,E2 -30329.998} C_VEL
LIN {X 0,Y 27.624,Z 549.495,A -85,B 0,C 180,E1 -30344.738,E2 -30344.738} C_VEL
LIN {X 0,Y 33.086,Z 551.355,A -85,B 0,C 180,E1 -30369.585,E2 -30369.585} C_VEL
LIN {X 0,Y 42.597,Z 551.621,A -85,B 0,C 180,E1 -30385.58,E2 -30385.58} C_VEL
LIN {X 0,Y 48.27,Z 551.282,A -85,B 0,C 180,E1 -30390.877,E2 -30390.877} C_VEL
LIN {X 0,Y 60.483,Z 549.377,A -85,B 0,C 180,E1 -30398.368,E2 -30398.368} C_VEL
LIN {X 0,Y 73.355,Z 545.83,A -85,B 0,C 180,E1 -30403.349,E2 -30403.349} C_VEL
LIN {X 0,Y 83.299,Z 542.117,A -85,B 0,C 180,E1 -30405.992,E2 -30405.992} C_VEL
LIN {X 0,Y 93.413,Z 537.331,A -85,B 0,C 180,E1 -30407.975,E2 -30407.975} C_VEL
LIN {X 0,Y 93.103,Z 537.484,A -85,B 0,C 180,E1 -30408.908,E2 -30408.908} C_VEL
LIN {X 0,Y 81.59,Z 542.788,A -85,B 0,C 180,E1 -30411.341,E2 -30411.341} C_VEL
LIN {X 0,Y 70.605,Z 546.603,A -85,B 0,C 180,E1 -30414.498,E2 -30414.498} C_VEL
LIN {X 0,Y 57.698,Z 549.598,A -85,B 0,C 180,E1 -30420.002,E2 -30420.002} C_VEL
LIN {X 0,Y 49.41,Z 550.803,A -85,B 0,C 180,E1 -30425.343,E2 -30425.343} C_VEL
LIN {X 0,Y 37.791,Z 551.075,A -85,B 0,C 180,E1 -30437.898,E2 -30437.898} C_VEL
LIN {X 0,Y 33.401,Z 550.857,A -85,B 0,C 180,E1 -30444.281,E2 -30444.281} C_VEL
LIN {X 0,Y 25.791,Z 549.801,A -85,B 0,C 180,E1 -30456.599,E2 -30456.599} C_VEL
LIN {X 0,Y 20.866,Z 548.32,A -85,B 0,C 180,E1 -30471.795,E2 -30471.795} C_VEL
LIN {X 0,Y 19.265,Z 546.825,A -85,B 0,C 180,E1 -30487.684,E2 -30487.684} C_VEL
LIN {X 0,Y 19.342,Z 546.245,A -85,B 0,C 180,E1 -30493.326,E2 -30493.326} C_VEL
LIN {X 0,Y 22.748,Z 542.946,A -85,B 0,C 180,E1 -30519.3,E2 -30519.3} C_VEL
LIN {X 0,Y 29.717,Z 538.079,A -85,B 0,C 180,E1 -30538.231,E2 -30538.231} C_VEL
LIN {X 0,Y 38.46,Z 531.781,A -85,B 0,C 180,E1 -30549.762,E2 -30549.762} C_VEL
LIN {X 0,Y 46.424,Z 525.375,A -85,B 0,C 180,E1 -30555.98,E2 -30555.98} C_VEL
LIN {X 0,Y 54.759,Z 517.596,A -85,B 0,C 180,E1 -30560.361,E2 -30560.361} C_VEL
LIN {X 0,Y 62.348,Z 509.198,A -85,B 0,C 180,E1 -30563.432,E2 -30563.432} C_VEL
LIN {X 0,Y 69.309,Z 500.161,A -85,B 0,C 180,E1 -30565.477,E2 -30565.477} C_VEL
LIN {X 0,Y 75.403,Z 490.635,A -85,B 0,C 180,E1 -30567.02,E2 -30567.02} C_VEL
LIN {X 0,Y 80.375,Z 481.221,A -85,B 0,C 180,E1 -30568.156,E2 -30568.156} C_VEL
LIN {X 0,Y 84.705,Z 471.127,A -85,B 0,C 180,E1 -30569.006,E2 -30569.006} C_VEL
LIN {X 0,Y 88.271,Z 460.245,A -85,B 0,C 180,E1 -30569.721,E2 -30569.721} C_VEL
LIN {X 0,Y 90.848,Z 449.615,A -85,B 0,C 180,E1 -30570.1,E2 -30570.1} C_VEL
LIN {X 0,Y 92.565,Z 438.791,A -85,B 0,C 180,E1 -30570.447,E2 -30570.447} C_VEL
LIN {X 0,Y 91.482,Z 434.759,A -85,B 0,C 180,E1 -30574.434,E2 -30574.434} C_VEL
LIN {X 0,Y 90.624,Z 431.777,A -85,B 0,C 180,E1 -30578.66,E2 -30578.66} C_VEL
LIN {X 0,Y 90.271,Z 430.616,A -85,B 0,C 180,E1 -30581.052,E2 -30581.052} C_VEL
LIN {X 0,Y 90.023,Z 428.164,A -85,B 0,C 180,E1 -30587.733,E2 -30587.733} C_VEL
LIN {X 0,Y 90.089,Z 428.237,A -85,B 0,C 180,E1 -30590.667,E2 -30590.667} C_VEL
LIN {X 0,Y 90.523,Z 430.64,A -85,B 0,C 180,E1 -30596.05,E2 -30596.05} C_VEL
LIN {X 0,Y 91.432,Z 434.39,A -85,B 0,C 180,E1 -30601.107,E2 -30601.107} C_VEL
LIN {X 0,Y 92.602,Z 438.834,A -85,B 0,C 180,E1 -30605.468,E2 -30605.468} C_VEL
LIN {X 0,Y 90.17,Z 453.752,A -85,B 0,C 180,E1 -30605.992,E2 -30605.992} C_VEL
LIN {X 0,Y 86.316,Z 467.19,A -85,B 0,C 180,E1 -30606.608,E2 -30606.608} C_VEL
LIN {X 0,Y 82.353,Z 477.362,A -85,B 0,C 180,E1 -30607.213,E2 -30607.213} C_VEL
LIN {X 0,Y 77.243,Z 487.884,A -85,B 0,C 180,E1 -30608.321,E2 -30608.321} C_VEL
LIN {X 0,Y 72.114,Z 496.452,A -85,B 0,C 180,E1 -30609.334,E2 -30609.334} C_VEL
LIN {X 0,Y 65.377,Z 505.945,A -85,B 0,C 180,E1 -30611.204,E2 -30611.204} C_VEL
LIN {X 0,Y 57.908,Z 514.769,A -85,B 0,C 180,E1 -30613.847,E2 -30613.847} C_VEL
LIN {X 0,Y 51.347,Z 521.41,A -85,B 0,C 180,E1 -30616.641,E2 -30616.641} C_VEL
LIN {X 0,Y 43.433,Z 528.389,A -85,B 0,C 180,E1 -30621.496,E2 -30621.496} C_VEL
LIN {X 0,Y 35.915,Z 534.207,A -85,B 0,C 180,E1 -30628.285,E2 -30628.285} C_VEL
LIN {X 0,Y 27.875,Z 539.82,A -85,B 0,C 180,E1 -30640.851,E2 -30640.851} C_VEL
LIN {X 0,Y 22.019,Z 544.224,A -85,B 0,C 180,E1 -30661.393,E2 -30661.393} C_VEL
LIN {X 0,Y 19.948,Z 547.522,A -85,B 0,C 180,E1 -30689.998,E2 -30689.998} C_VEL
LIN {X 0,Y 20.849,Z 549.086,A -85,B 0,C 180,E1 -30709.698,E2 -30709.698} C_VEL
LIN {X 0,Y 27.966,Z 551.145,A -85,B 0,C 180,E1 -30738.928,E2 -30738.928} C_VEL
LIN {X 0,Y 39.023,Z 551.587,A -85,B 0,C 180,E1 -30754.22,E2 -30754.22} C_VEL
LIN {X 0,Y 51.664,Z 550.536,A -85,B 0,C 180,E1 -30762.217,E2 -30762.217} C_VEL
LIN {X 0,Y 58.241,Z 549.562,A -85,B 0,C 180,E1 -30764.876,E2 -30764.876} C_VEL
LIN {X 0,Y 70.105,Z 546.712,A -85,B 0,C 180,E1 -30768.435,E2 -30768.435} C_VEL
LIN {X 0,Y 56.247,Z 549.75,A -85,B 0,C 180,E1 -30772.824,E2 -30772.824} C_VEL
LIN {X 0,Y 49.316,Z 550.716,A -85,B 0,C 180,E1 -30775.991,E2 -30775.991} C_VEL
LIN {X 0,Y 35.369,Z 551.258,A -85,B 0,C 180,E1 -30786.534,E2 -30786.534} C_VEL
LIN {X 0,Y 29.145,Z 550.876,A -85,B 0,C 180,E1 -30795.304,E2 -30795.304} C_VEL
LIN {X 0,Y 20.305,Z 548.539,A -85,B 0,C 180,E1 -30826.196,E2 -30826.196} C_VEL
LIN {X 0,Y 19.342,Z 546.245,A -85,B 0,C 180,E1 -30853.326,E2 -30853.326} C_VEL
LIN {X 0,Y 20.102,Z 544.459,A -85,B 0,C 180,E1 -30869.458,E2 -30869.458} C_VEL
LIN {X 0,Y 21.28,Z 542.462,A -85,B 0,C 180,E1 -30884.589,E2 -30884.589} C_VEL
LIN {X 0,Y 26.305,Z 537.617,A -85,B 0,C 180,E1 -30908.465,E2 -30908.465} C_VEL
LIN {X 0,Y 30.325,Z 534.733,A -85,B 0,C 180,E1 -30915.474,E2 -30915.474} C_VEL
LIN {X 0,Y 31.869,Z 533.744,A -85,B 0,C 180,E1 -30916.998,E2 -30916.998} C_VEL
LIN {X 0,Y 43.349,Z 525.342,A -85,B 0,C 180,E1 -30924.16,E2 -30924.16} C_VEL
LIN {X 0,Y 52.303,Z 517.362,A -85,B 0,C 180,E1 -30927.486,E2 -30927.486} C_VEL
LIN {X 0,Y 59.149,Z 510.177,A -85,B 0,C 180,E1 -30929.479,E2 -30929.479} C_VEL
LIN {X 0,Y 66.29,Z 501.332,A -85,B 0,C 180,E1 -30931.006,E2 -30931.006} C_VEL
LIN {X 0,Y 72.432,Z 492.23,A -85,B 0,C 180,E1 -30932.107,E2 -30932.107} C_VEL
LIN {X 0,Y 78.318,Z 481.463,A -85,B 0,C 180,E1 -30933.063,E2 -30933.063} C_VEL
LIN {X 0,Y 82.495,Z 472.066,A -85,B 0,C 180,E1 -30933.647,E2 -30933.647} C_VEL
LIN {X 0,Y 86.416,Z 460.452,A -85,B 0,C 180,E1 -30934.208,E2 -30934.208} C_VEL
LIN {X 0,Y 89.037,Z 449.798,A -85,B 0,C 180,E1 -30934.489,E2 -30934.489} C_VEL
LIN {X 0,Y 90.305,Z 442.461,A -85,B 0,C 180,E1 -30934.717,E2 -30934.717} C_VEL
LIN {X 0,Y 89.525,Z 438.857,A -85,B 0,C 180,E1 -30939.26,E2 -30939.26} C_VEL
LIN {X 0,Y 89.183,Z 437.439,A -85,B 0,C 180,E1 -30942.113,E2 -30942.113} C_VEL
LIN {X 0,Y 89.047,Z 435.479,A -85,B 0,C 180,E1 -30947.597,E2 -30947.597} C_VEL
LIN {X 0,Y 89.126,Z 435.913,A -85,B 0,C 180,E1 -30951.496,E2 -30951.496} C_VEL
LIN {X 0,Y 89.379,Z 437.484,A -85,B 0,C 180,E1 -30954.936,E2 -30954.936} C_VEL
LIN {X 0,Y 90.076,Z 441.09,A -85,B 0,C 180,E1 -30959.718,E2 -30959.718} C_VEL
LIN {X 0,Y 90.356,Z 442.555,A -85,B 0,C 180,E1 -30961.252,E2 -30961.252} C_VEL
LIN {X 0,Y 87.795,Z 455.839,A -85,B 0,C 180,E1 -30961.67,E2 -30961.67} C_VEL
LIN {X 0,Y 84.389,Z 467.274,A -85,B 0,C 180,E1 -30962.022,E2 -30962.022} C_VEL
LIN {X 0,Y 80.891,Z 476.286,A -85,B 0,C 180,E1 -30962.348,E2 -30962.348} C_VEL
LIN {X 0,Y 75.665,Z 486.994,A -85,B 0,C 180,E1 -30963.138,E2 -30963.138} C_VEL
LIN {X 0,Y 69.566,Z 496.938,A -85,B 0,C 180,E1 -30963.932,E2 -30963.932} C_VEL
LIN {X 0,Y 63.509,Z 505.312,A -85,B 0,C 180,E1 -30965.145,E2 -30965.145} C_VEL
LIN {X 0,Y 55.35,Z 514.636,A -85,B 0,C 180,E1 -30967.144,E2 -30967.144} C_VEL
LIN {X 0,Y 48.08,Z 521.656,A -85,B 0,C 180,E1 -30969.361,E2 -30969.361} C_VEL
LIN {X 0,Y 39.695,Z 528.576,A -85,B 0,C 180,E1 -30973.147,E2 -30973.147} C_VEL
LIN {X 0,Y 33.138,Z 533.3,A -85,B 0,C 180,E1 -30977.371,E2 -30977.371} C_VEL
LIN {X 0,Y 23.833,Z 539.109,A -85,B 0,C 180,E1 -30987.788,E2 -30987.788} C_VEL
LIN {X 0,Y 16.15,Z 543.66,A -85,B 0,C 180,E1 -31009.246,E2 -31009.246} C_VEL
LIN {X 0,Y 12.874,Z 547.078,A -85,B 0,C 180,E1 -31049.997,E2 -31049.997} C_VEL
LIN {X 0,Y 14.383,Z 548.661,A -85,B 0,C 180,E1 -31079.247,E2 -31079.247} C_VEL
LIN {X 0,Y 23.9,Z 550.859,A -85,B 0,C 180,E1 -31111.904,E2 -31111.904} C_VEL
LIN {X 0,Y 36.499,Z 551.541,A -85,B 0,C 180,E1 -31124.311,E2 -31124.311} C_VEL
LIN {X 0,Y 43.177,Z 551.214,A -85,B 0,C 180,E1 -31127.582,E2 -31127.582} C_VEL
LIN {X 0,Y 42.87,Z 551.207,A -85,B 0,C 180,E1 -31129.615,E2 -31129.615} C_VEL
LIN {X 0,Y 35.366,Z 551.448,A -85,B 0,C 180,E1 -31133.513,E2 -31133.513} C_VEL
LIN {X 0,Y 27.565,Z 551.036,A -85,B 0,C 180,E1 -31140.004,E2 -31140.004} C_VEL
LIN {X 0,Y 15.229,Z 548.902,A -85,B 0,C 180,E1 -31167.491,E2 -31167.491} C_VEL
LIN {X 0,Y 12.324,Z 545.934,A -85,B 0,C 180,E1 -31217.163,E2 -31217.163} C_VEL
LIN {X 0,Y 17.612,Z 542.238,A -85,B 0,C 180,E1 -31253.522,E2 -31253.522} C_VEL
LIN {X 0,Y 23.396,Z 538.998,A -85,B 0,C 180,E1 -31266.928,E2 -31266.928} C_VEL
LIN {X 0,Y 31.869,Z 533.744,A -85,B 0,C 180,E1 -31276.998,E2 -31276.998} C_VEL
LIN {X 0,Y 36.21,Z 530.678,A -85,B 0,C 180,E1 -31281.318,E2 -31281.318} C_VEL
LIN {X 0,Y 42.594,Z 525.027,A -85,B 0,C 180,E1 -31288.703,E2 -31288.703} C_VEL
LIN {X 0,Y 49.02,Z 518.856,A -85,B 0,C 180,E1 -31294.11,E2 -31294.11} C_VEL
LIN {X 0,Y 53.137,Z 514.678,A -85,B 0,C 180,E1 -31295.572,E2 -31295.572} C_VEL
LIN {X 0,Y 60.297,Z 506.808,A -85,B 0,C 180,E1 -31296.619,E2 -31296.619} C_VEL
LIN {X 0,Y 65.781,Z 499.814,A -85,B 0,C 180,E1 -31297.146,E2 -31297.146} C_VEL
LIN {X 0,Y 71.504,Z 491.264,A -85,B 0,C 180,E1 -31297.691,E2 -31297.691} C_VEL
LIN {X 0,Y 76.514,Z 482.299,A -85,B 0,C 180,E1 -31298.154,E2 -31298.154} C_VEL
LIN {X 0,Y 81.466,Z 471.163,A -85,B 0,C 180,E1 -31298.545,E2 -31298.545} C_VEL
LIN {X 0,Y 85.16,Z 460.233,A -85,B 0,C 180,E1 -31298.875,E2 -31298.875} C_VEL
LIN {X 0,Y 87.835,Z 449.301,A -85,B 0,C 180,E1 -31299.002,E2 -31299.002} C_VEL
LIN {X 0,Y 88.293,Z 446.59,A -85,B 0,C 180,E1 -31299.144,E2 -31299.144} C_VEL
LIN {X 0,Y 88.045,Z 444.345,A -85,B 0,C 180,E1 -31302.882,E2 -31302.882} C_VEL
LIN {X 0,Y 88.04,Z 442.786,A -85,B 0,C 180,E1 -31307.453,E2 -31307.453} C_VEL
LIN {X 0,Y 88.112,Z 443.115,A -85,B 0,C 180,E1 -31311.398,E2 -31311.398} C_VEL
LIN {X 0,Y 88.199,Z 444.643,A -85,B 0,C 180,E1 -31314.307,E2 -31314.307} C_VEL
LIN {X 0,Y 88.36,Z 446.557,A -85,B 0,C 180,E1 -31316.858,E2 -31316.858} C_VEL
LIN {X 0,Y 86.371,Z 456.164,A -85,B 0,C 180,E1 -31317.106,E2 -31317.106} C_VEL
LIN {X 0,Y 83.093,Z 467.038,A -85,B 0,C 180,E1 -31317.255,E2 -31317.255} C_VEL
LIN {X 0,Y 79.015,Z 477.234,A -85,B 0,C 180,E1 -31317.408,E2 -31317.408} C_VEL
LIN {X 0,Y 73.846,Z 487.516,A -85,B 0,C 180,E1 -31317.869,E2 -31317.869} C_VEL
LIN {X 0,Y 67.679,Z 497.336,A -85,B 0,C 180,E1 -31318.197,E2 -31318.197} C_VEL
LIN {X 0,Y 61.508,Z 505.618,A -85,B 0,C 180,E1 -31318.862,E2 -31318.862} C_VEL
LIN {X 0,Y 54.724,Z 513.343,A -85,B 0,C 180,E1 -31319.742,E2 -31319.742} C_VEL
LIN {X 0,Y 45.693,Z 521.837,A -85,B 0,C 180,E1 -31321.188,E2 -31321.188} C_VEL
LIN {X 0,Y 36.959,Z 528.699,A -85,B 0,C 180,E1 -31323.295,E2 -31323.295} C_VEL
LIN {X 0,Y 28.287,Z 534.406,A -85,B 0,C 180,E1 -31326.356,E2 -31326.356} C_VEL
LIN {X 0,Y 18.112,Z 539.937,A -85,B 0,C 180,E1 -31334.046,E2 -31334.046} C_VEL
LIN {X 0,Y 8.878,Z 544.254,A -85,B 0,C 180,E1 -31357.658,E2 -31357.658} C_VEL
LIN {X 0,Y 5.784,Z 546.536,A -85,B 0,C 180,E1 -31409.993,E2 -31409.993} C_VEL
LIN {X 0,Y 14.864,Z 549.66,A -85,B 0,C 180,E1 -31481.018,E2 -31481.018} C_VEL
LIN {X 0,Y 18.034,Z 550.077,A -85,B 0,C 180,E1 -31490.44,E2 -31490.44} C_VEL
LIN {X 0,Y 11.756,Z 548.957,A -85,B 0,C 180,E1 -31500.009,E2 -31500.009} C_VEL
LIN {X 0,Y 5.232,Z 546.841,A -85,B 0,C 180,E1 -31547.817,E2 -31547.817} C_VEL
LIN {X 0,Y 11.04,Z 543.047,A -85,B 0,C 180,E1 -31629.542,E2 -31629.542} C_VEL
LIN {X 0,Y 21.521,Z 538.045,A -85,B 0,C 180,E1 -31644.732,E2 -31644.732} C_VEL
LIN {X 0,Y 32.249,Z 531.702,A -85,B 0,C 180,E1 -31650.661,E2 -31650.661} C_VEL
LIN {X 0,Y 41.285,Z 525.241,A -85,B 0,C 180,E1 -31653.346,E2 -31653.346} C_VEL
LIN {X 0,Y 49.955,Z 517.803,A -85,B 0,C 180,E1 -31655.033,E2 -31655.033} C_VEL
LIN {X 0,Y 53.137,Z 514.678,A -85,B 0,C 180,E1 -31655.572,E2 -31655.572} C_VEL
LIN {X 0,Y 57.102,Z 510.487,A -85,B 0,C 180,E1 -31656.822,E2 -31656.822} C_VEL
LIN {X 0,Y 62.87,Z 503.14,A -85,B 0,C 180,E1 -31660.135,E2 -31660.135} C_VEL
LIN {X 0,Y 68.172,Z 495.376,A -85,B 0,C 180,E1 -31662.838,E2 -31662.838} C_VEL
LIN {X 0,Y 71.248,Z 490.308,A -85,B 0,C 180,E1 -31663.364,E2 -31663.364} C_VEL
LIN {X 0,Y 76.11,Z 481.474,A -85,B 0,C 180,E1 -31663.45,E2 -31663.45} C_VEL
LIN {X 0,Y 80.619,Z 471.347,A -85,B 0,C 180,E1 -31663.525,E2 -31663.525} C_VEL
LIN {X 0,Y 84.241,Z 460.819,A -85,B 0,C 180,E1 -31663.614,E2 -31663.614} C_VEL
LIN {X 0,Y 86.689,Z 451.412,A -85,B 0,C 180,E1 -31663.657,E2 -31663.657} C_VEL
LIN {X 0,Y 86.775,Z 449.833,A -85,B 0,C 180,E1 -31667.949,E2 -31667.949} C_VEL
LIN {X 0,Y 86.823,Z 450.188,A -85,B 0,C 180,E1 -31671.145,E2 -31671.145} C_VEL
LIN {X 0,Y 86.799,Z 450.904,A -85,B 0,C 180,E1 -31672.281,E2 -31672.281} C_VEL
LIN {X 0,Y 83.241,Z 464.382,A -85,B 0,C 180,E1 -31672.363,E2 -31672.363} C_VEL
LIN {X 0,Y 78.577,Z 476.379,A -85,B 0,C 180,E1 -31672.277,E2 -31672.277} C_VEL
LIN {X 0,Y 73.569,Z 486.473,A -85,B 0,C 180,E1 -31672.362,E2 -31672.362} C_VEL
LIN {X 0,Y 67.389,Z 496.466,A -85,B 0,C 180,E1 -31672.206,E2 -31672.206} C_VEL
LIN {X 0,Y 60.29,Z 505.901,A -85,B 0,C 180,E1 -31672.246,E2 -31672.246} C_VEL
LIN {X 0,Y 52.758,Z 514.234,A -85,B 0,C 180,E1 -31672.343,E2 -31672.343} C_VEL
LIN {X 0,Y 44.326,Z 522.007,A -85,B 0,C 180,E1 -31672.291,E2 -31672.291} C_VEL
LIN {X 0,Y 35.465,Z 528.821,A -85,B 0,C 180,E1 -31672.252,E2 -31672.252} C_VEL
LIN {X 0,Y 28.395,Z 533.5,A -85,B 0,C 180,E1 -31671.918,E2 -31671.918} C_VEL
LIN {X 0,Y 17.782,Z 539.212,A -85,B 0,C 180,E1 -31671.152,E2 -31671.152} C_VEL
LIN {X 0,Y 14.252,Z 540.74,A -85,B 0,C 180,E1 -31670.497,E2 -31670.497} C_VEL
LIN {X 0,Y 14.523,Z 540.608,A -85,B 0,C 180,E1 -31665.441,E2 -31665.441} C_VEL
LIN {X 0,Y 21.96,Z 537,A -85,B 0,C 180,E1 -31663.768,E2 -31663.768} C_VEL
LIN {X 0,Y 31.178,Z 531.636,A -85,B 0,C 180,E1 -31663.341,E2 -31663.341} C_VEL
LIN {X 0,Y 40.371,Z 525.143,A -85,B 0,C 180,E1 -31663.236,E2 -31663.236} C_VEL
LIN {X 0,Y 48.587,Z 518.206,A -85,B 0,C 180,E1 -31663.182,E2 -31663.182} C_VEL
LIN {X 0,Y 56.856,Z 509.807,A -85,B 0,C 180,E1 -31663.335,E2 -31663.335} C_VEL
LIN {X 0,Y 64.196,Z 500.848,A -85,B 0,C 180,E1 -31663.323,E2 -31663.323} C_VEL
LIN {X 0,Y 70.595,Z 491.413,A -85,B 0,C 180,E1 -31663.378,E2 -31663.378} C_VEL
LIN {X 0,Y 71.248,Z 490.308,A -85,B 0,C 180,E1 -31663.364,E2 -31663.364} C_VEL
LIN {X 0,Y 74.969,Z 491.325,A -85,B 0,C 180,E1 -31663.291,E2 -31663.291} C_VEL
LIN {X 0,Y 74.969,Z 600,A -85,B 0,C 180,E1 -31663.291,E2 -31663.291} C_VEL
LIN {X 0,Y 74.969,Z 600,A -85,B 0,C 180,E1 -31663.291,E2 -31663.291}

QRS_NEXT_CUT()

QRS_NEXT()
QRS_HOME()

END
